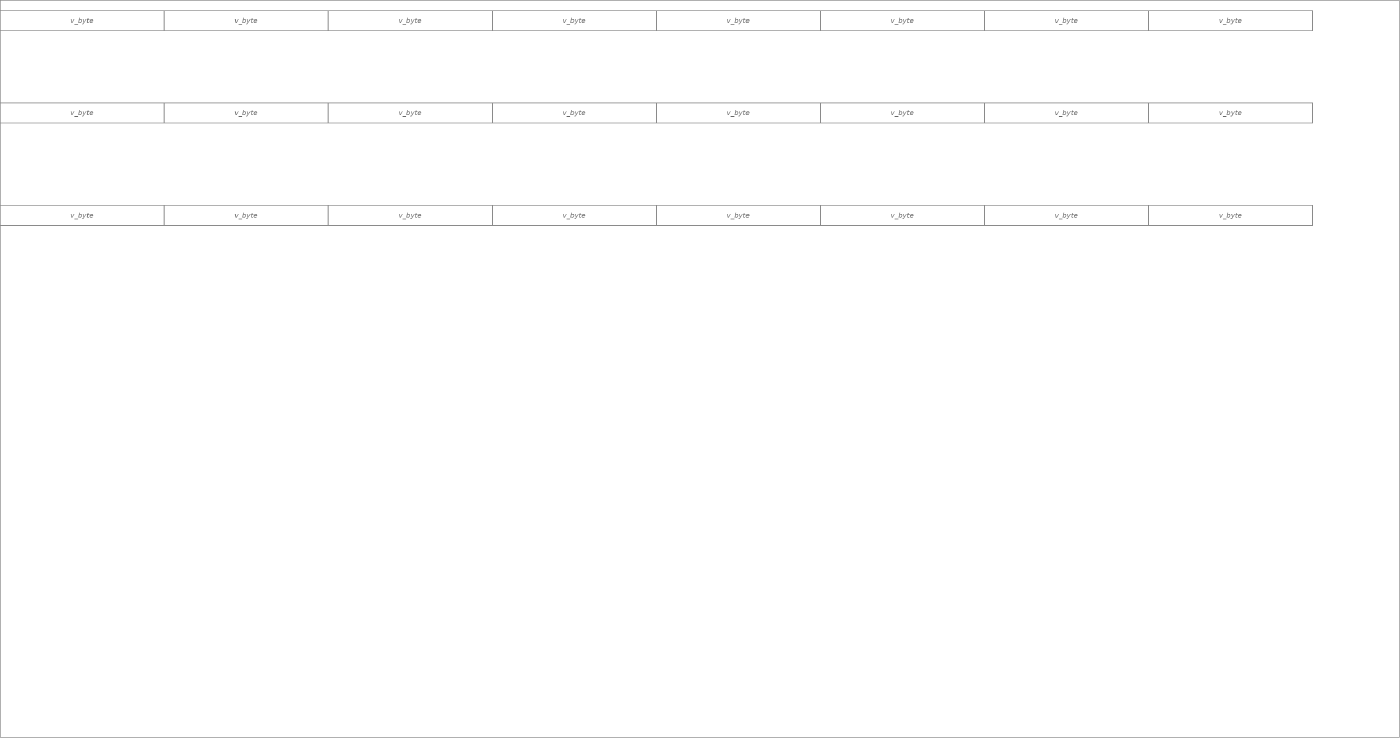
VISUALIZATION visu_MLC  // 2048x1080
    Frame (0,15 240x30)
        shows v_byte(iNum := GVL.ibyteNum[1])
    Frame (0,300 240x30)
        shows v_byte(iNum := GVL.ibyteNum[17])
    Frame (240,300 240x30)
        shows v_byte(iNum := GVL.ibyteNum[18])
    Frame (480,300 240x30)
        shows v_byte(iNum := GVL.ibyteNum[19])
    Frame (720,300 240x30)
        shows v_byte(iNum := GVL.ibyteNum[20])
    Frame (960,300 240x30)
        shows v_byte(iNum := GVL.ibyteNum[21])
    Frame (1200,300 240x30)
        shows v_byte(iNum := GVL.ibyteNum[22])
    Frame (1440,300 240x30)
        shows v_byte(iNum := GVL.ibyteNum[23])
    Frame (1680,300 240x30)
        shows v_byte(iNum := GVL.ibyteNum[24])
    Frame (0,150 240x30)
        shows v_byte(iNum := GVL.ibyteNum[9])
    Frame (240,150 240x30)
        shows v_byte(iNum := GVL.ibyteNum[10])
    Frame (480,150 240x30)
        shows v_byte(iNum := GVL.ibyteNum[11])
    Frame (720,150 240x30)
        shows v_byte(iNum := GVL.ibyteNum[12])
    Frame (960,150 240x30)
        shows v_byte(iNum := GVL.ibyteNum[13])
    Frame (1200,150 240x30)
        shows v_byte(iNum := GVL.ibyteNum[14])
    Frame (1440,150 240x30)
        shows v_byte(iNum := GVL.ibyteNum[15])
    Frame (1680,150 240x30)
        shows v_byte(iNum := GVL.ibyteNum[16])
    Frame (240,15 240x30)
        shows v_byte(iNum := GVL.ibyteNum[2])
    Frame (480,15 240x30)
        shows v_byte(iNum := GVL.ibyteNum[3])
    Frame (720,15 240x30)
        shows v_byte(iNum := GVL.ibyteNum[4])
    Frame (960,15 240x30)
        shows v_byte(iNum := GVL.ibyteNum[5])
    Frame (1200,15 240x30)
        shows v_byte(iNum := GVL.ibyteNum[6])
    Frame (1440,15 240x30)
        shows v_byte(iNum := GVL.ibyteNum[7])
    Frame (1680,15 240x30)
        shows v_byte(iNum := GVL.ibyteNum[8])
END_VISUALIZATION

(* stored: Version 1.1.0.1, ProductVersion 3.1.4024.12
   Visu visu_MLC: Id {967a5305-adcb-48b3-aa96-204a00315718} *)
